// TIA Portal V15.1 export
// export: Created 2024-06-21T08:41:21.5469996Z, ExportSetting WithDefaults, DisplayName Totally Integrated Automation Portal, DisplayVersion V15.1 Update 5, DisplayName TIA Portal Openness, DisplayVersion V15.1 Update 5, DisplayName SINAMICS Startdrive Advanced, DisplayVersion V15.1, DisplayName G130, G150, S120, S150, SINAMICS MV, S210, DisplayVersion V15.1, DisplayName G110M, G120, G120C, G120D, G120P, DisplayVersion V15.1, DisplayName STEP 7 Professional, DisplayVersion V15.1 Update 5, DisplayName STEP 7 Safety, DisplayVersion V15.1, DisplayName WinCC Professional, DisplayVersion V15.1 Update 5, DisplayName SIMATIC Visualization Architect, DisplayVersion V15.1
FUNCTION "209220ZS01AEAK" : Void   // FC371, FBD
TITLE = 209220ZS01AEAK
{ S7_Optimized_Access := 'TRUE' }
AUTHOR : VCC
VERSION : 0.1
// stored: AutoNumber false, IsIECCheckEnabled false, SetENOAutomatically False, UDAEnableTagReadback false
   VAR_OUTPUT
      O_AlarmA : Bool;   // Alarm A
      O_AlarmB : Bool;   // Alarm B
      O_AlarmC : Bool;   // Alarm C
      O_AlarmD : Bool;   // Alarm D
      O_AlarmABCondition : Bool;   // Alarm AB condition
      H_IAnim : Word;   // For animation of icon
   END_VAR
BEGIN

REGION Network 1: **** --------------------- AE01 --------------------- ****
END_REGION

REGION Network 2: **** 2.2 Alarms - Alarm generation **** AE01E3FS10 // CH1 - 24VDC Fuse - ModeZone220 - Switch / Busnode 220AX01 & 220AS10
   // 24VDC Fuse - ModeZone220 - Switch / Busnode 220AX01 & 220AS10
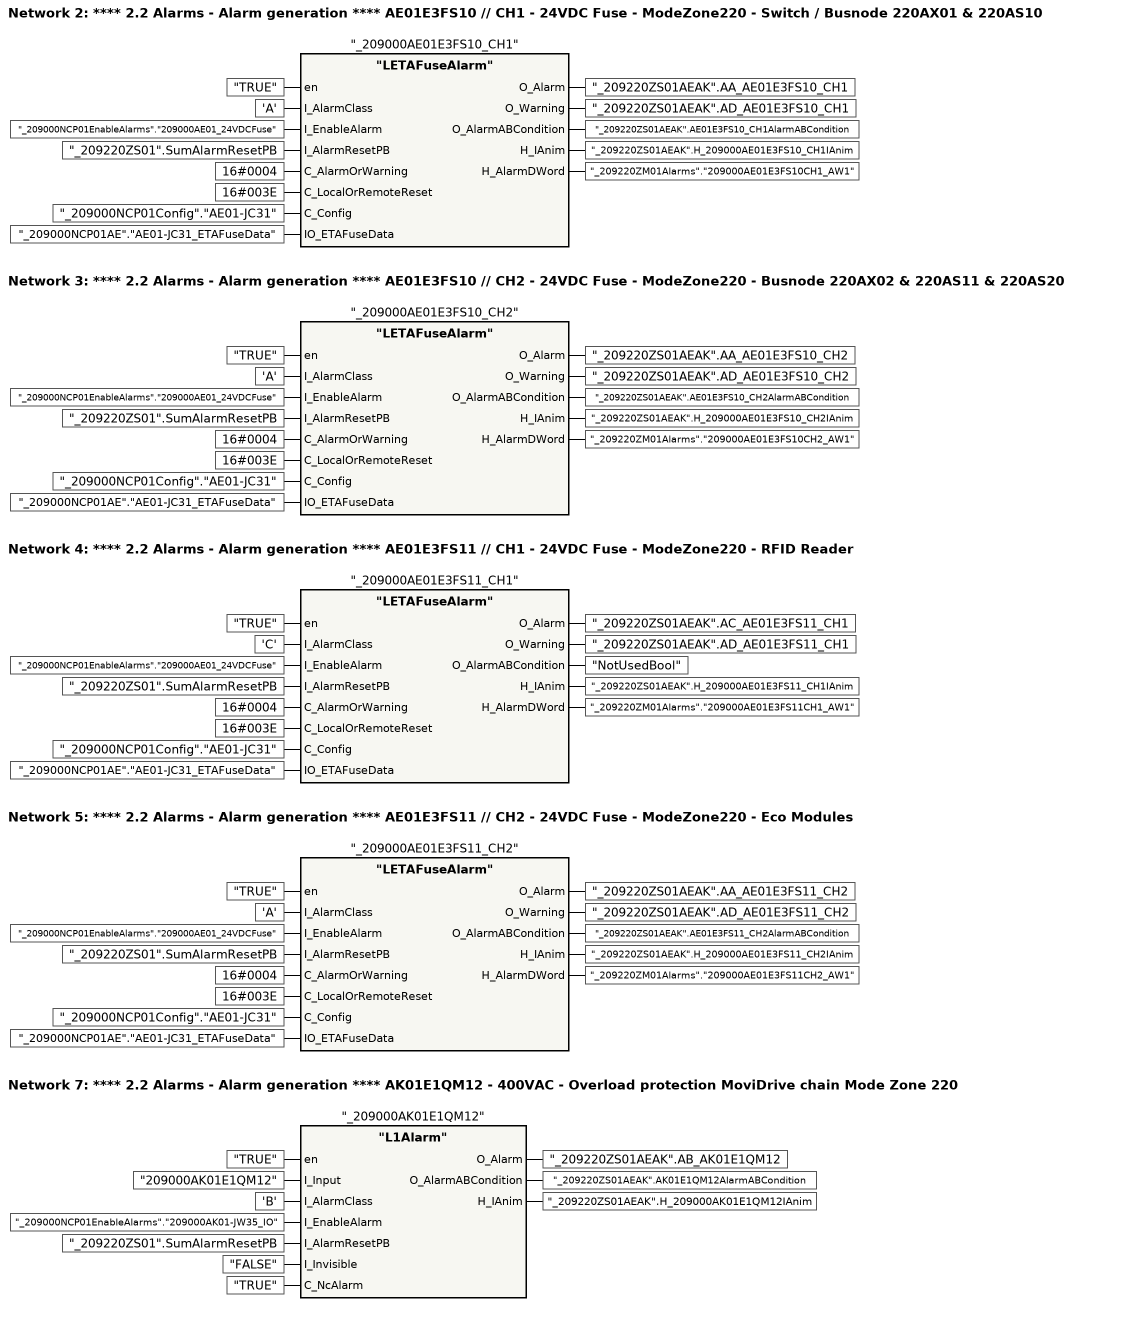
   IF "TRUE" THEN
       "_209000AE01E3FS10_CH1"(I_AlarmClass := 'A',   // "LETAFuseAlarm"
                               I_EnableAlarm := "_209000NCP01EnableAlarms"."209000AE01_24VDCFuse",
                               I_AlarmResetPB := "_209220ZS01".SumAlarmResetPB,
                               C_AlarmOrWarning := 16#0004,
                               C_LocalOrRemoteReset := 16#003E,
                               C_Config := "_209000NCP01Config"."AE01-JC31",
                               IO_ETAFuseData := "_209000NCP01AE"."AE01-JC31_ETAFuseData",
                               O_Alarm => "_209220ZS01AEAK".AA_AE01E3FS10_CH1,
                               O_Warning => "_209220ZS01AEAK".AD_AE01E3FS10_CH1,
                               O_AlarmABCondition => "_209220ZS01AEAK".AE01E3FS10_CH1AlarmABCondition,
                               H_IAnim => "_209220ZS01AEAK".H_209000AE01E3FS10_CH1IAnim,
                               H_AlarmDWord => "_209220ZM01Alarms"."209000AE01E3FS10CH1_AW1");
   END_IF;
END_REGION

REGION Network 3: **** 2.2 Alarms - Alarm generation **** AE01E3FS10 // CH2 - 24VDC Fuse - ModeZone220 - Busnode 220AX02 & 220AS11 & 220AS20
   // 24VDC Fuse - ModeZone220 - Busnode 220AX02 & 220AS11 & 220AS20
   IF "TRUE" THEN
       "_209000AE01E3FS10_CH2"(I_AlarmClass := 'A',   // "LETAFuseAlarm"
                               I_EnableAlarm := "_209000NCP01EnableAlarms"."209000AE01_24VDCFuse",
                               I_AlarmResetPB := "_209220ZS01".SumAlarmResetPB,
                               C_AlarmOrWarning := 16#0004,
                               C_LocalOrRemoteReset := 16#003E,
                               C_Config := "_209000NCP01Config"."AE01-JC31",
                               IO_ETAFuseData := "_209000NCP01AE"."AE01-JC31_ETAFuseData",
                               O_Alarm => "_209220ZS01AEAK".AA_AE01E3FS10_CH2,
                               O_Warning => "_209220ZS01AEAK".AD_AE01E3FS10_CH2,
                               O_AlarmABCondition => "_209220ZS01AEAK".AE01E3FS10_CH2AlarmABCondition,
                               H_IAnim => "_209220ZS01AEAK".H_209000AE01E3FS10_CH2IAnim,
                               H_AlarmDWord => "_209220ZM01Alarms"."209000AE01E3FS10CH2_AW1");
   END_IF;
END_REGION

REGION Network 4: **** 2.2 Alarms - Alarm generation **** AE01E3FS11 // CH1 - 24VDC Fuse - ModeZone220 - RFID Reader
   // 24VDC Fuse - ModeZone220 - RFID Reader
   IF "TRUE" THEN
       "_209000AE01E3FS11_CH1"(I_AlarmClass := 'C',   // "LETAFuseAlarm"
                               I_EnableAlarm := "_209000NCP01EnableAlarms"."209000AE01_24VDCFuse",
                               I_AlarmResetPB := "_209220ZS01".SumAlarmResetPB,
                               C_AlarmOrWarning := 16#0004,
                               C_LocalOrRemoteReset := 16#003E,
                               C_Config := "_209000NCP01Config"."AE01-JC31",
                               IO_ETAFuseData := "_209000NCP01AE"."AE01-JC31_ETAFuseData",
                               O_Alarm => "_209220ZS01AEAK".AC_AE01E3FS11_CH1,
                               O_Warning => "_209220ZS01AEAK".AD_AE01E3FS11_CH1,
                               O_AlarmABCondition => "NotUsedBool",
                               H_IAnim => "_209220ZS01AEAK".H_209000AE01E3FS11_CH1IAnim,
                               H_AlarmDWord => "_209220ZM01Alarms"."209000AE01E3FS11CH1_AW1");
   END_IF;
END_REGION

REGION Network 5: **** 2.2 Alarms - Alarm generation **** AE01E3FS11 // CH2 - 24VDC Fuse - ModeZone220 - Eco Modules
   // 24VDC Fuse - ModeZone220 - Eco Modules
   IF "TRUE" THEN
       "_209000AE01E3FS11_CH2"(I_AlarmClass := 'A',   // "LETAFuseAlarm"
                               I_EnableAlarm := "_209000NCP01EnableAlarms"."209000AE01_24VDCFuse",
                               I_AlarmResetPB := "_209220ZS01".SumAlarmResetPB,
                               C_AlarmOrWarning := 16#0004,
                               C_LocalOrRemoteReset := 16#003E,
                               C_Config := "_209000NCP01Config"."AE01-JC31",
                               IO_ETAFuseData := "_209000NCP01AE"."AE01-JC31_ETAFuseData",
                               O_Alarm => "_209220ZS01AEAK".AA_AE01E3FS11_CH2,
                               O_Warning => "_209220ZS01AEAK".AD_AE01E3FS11_CH2,
                               O_AlarmABCondition => "_209220ZS01AEAK".AE01E3FS11_CH2AlarmABCondition,
                               H_IAnim => "_209220ZS01AEAK".H_209000AE01E3FS11_CH2IAnim,
                               H_AlarmDWord => "_209220ZM01Alarms"."209000AE01E3FS11CH2_AW1");
   END_IF;
END_REGION

REGION Network 6: **** --------------------- AK01 --------------------- ****
END_REGION

REGION Network 7: **** 2.2 Alarms - Alarm generation **** AK01E1QM12 - 400VAC - Overload protection MoviDrive chain Mode Zone 220
   // 400VAC - Overload protection MoviDrive chain Mode Zone 220
   IF "TRUE" THEN
       "_209000AK01E1QM12"(I_Input := "209000AK01E1QM12",   // "L1Alarm"
                           I_AlarmClass := 'B',
                           I_EnableAlarm := "_209000NCP01EnableAlarms"."209000AK01-JW35_IO",
                           I_AlarmResetPB := "_209220ZS01".SumAlarmResetPB,
                           I_Invisible := "FALSE",
                           C_NcAlarm := "TRUE",
                           O_Alarm => "_209220ZS01AEAK".AB_AK01E1QM12,
                           O_AlarmABCondition => "_209220ZS01AEAK".AK01E1QM12AlarmABCondition,
                           H_IAnim => "_209220ZS01AEAK".H_209000AK01E1QM12IAnim);
   END_IF;
END_REGION

REGION Network 8: **** 2.2 Alarms - Alarm generation **** AK01E1QM13 - 400VAC - Overload protection MoviFit chain Mode Zone 220
   // 400VAC - Overload protection MoviFit chain Mode Zone 220
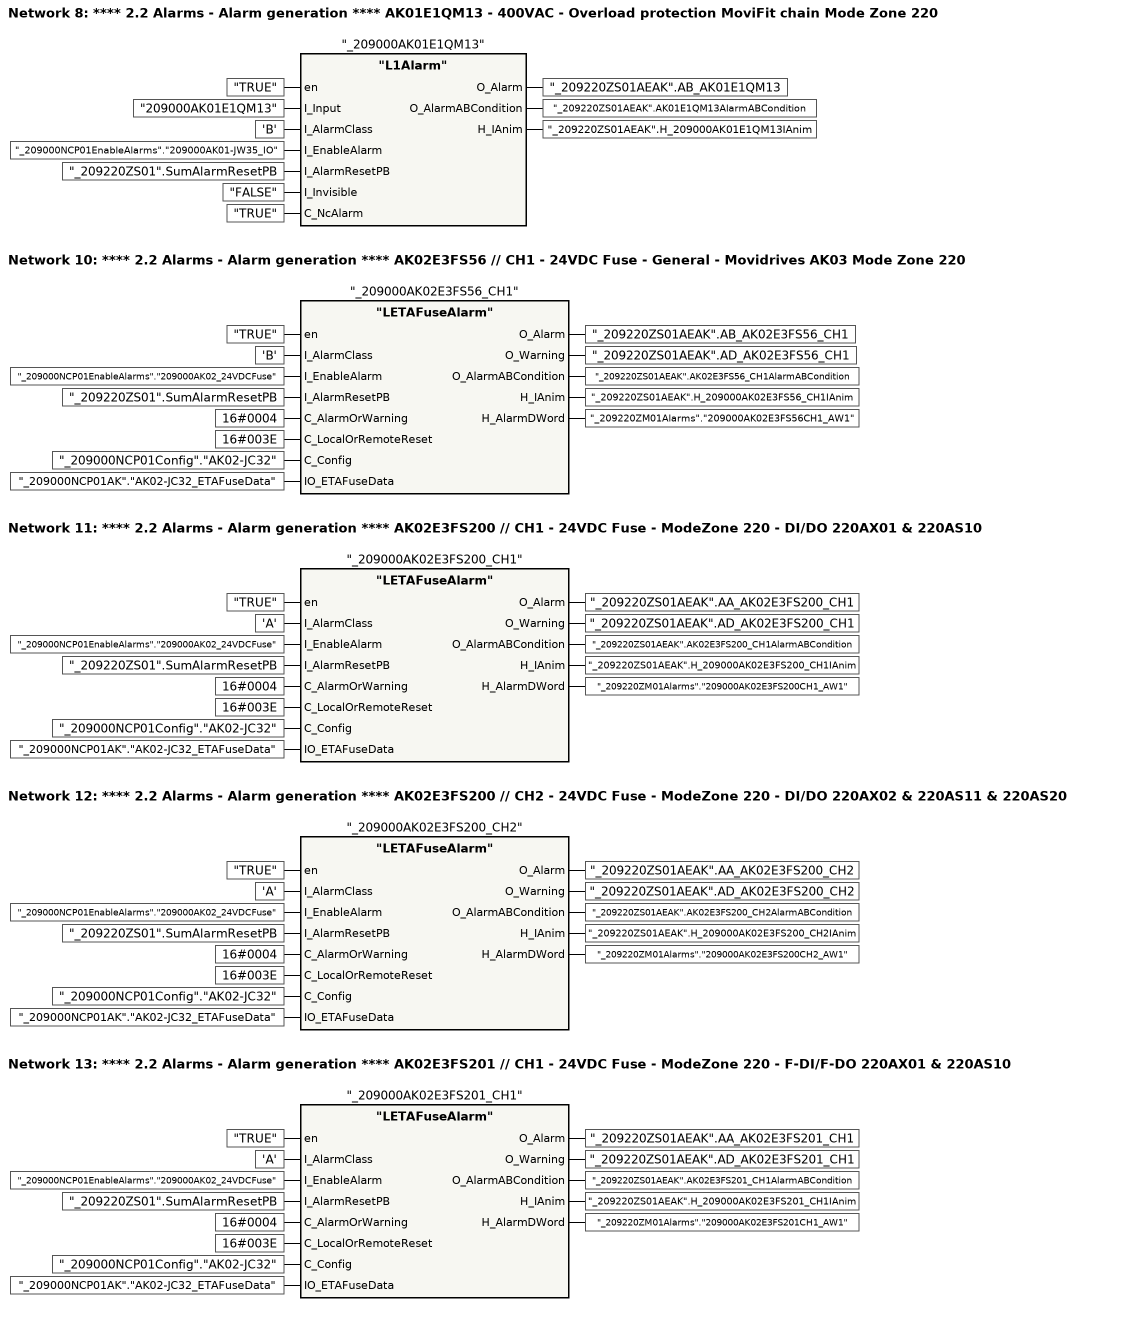
   IF "TRUE" THEN
       "_209000AK01E1QM13"(I_Input := "209000AK01E1QM13",   // "L1Alarm"
                           I_AlarmClass := 'B',
                           I_EnableAlarm := "_209000NCP01EnableAlarms"."209000AK01-JW35_IO",
                           I_AlarmResetPB := "_209220ZS01".SumAlarmResetPB,
                           I_Invisible := "FALSE",
                           C_NcAlarm := "TRUE",
                           O_Alarm => "_209220ZS01AEAK".AB_AK01E1QM13,
                           O_AlarmABCondition => "_209220ZS01AEAK".AK01E1QM13AlarmABCondition,
                           H_IAnim => "_209220ZS01AEAK".H_209000AK01E1QM13IAnim);
   END_IF;
END_REGION

REGION Network 9: **** --------------------- AK02 --------------------- ****
END_REGION

REGION Network 10: **** 2.2 Alarms - Alarm generation **** AK02E3FS56 // CH1 - 24VDC Fuse - General - Movidrives AK03 Mode Zone 220
   // 24VDC Fuse - General - Movidrives AK03 Mode Zone 220
   IF "TRUE" THEN
       "_209000AK02E3FS56_CH1"(I_AlarmClass := 'B',   // "LETAFuseAlarm"
                               I_EnableAlarm := "_209000NCP01EnableAlarms"."209000AK02_24VDCFuse",
                               I_AlarmResetPB := "_209220ZS01".SumAlarmResetPB,
                               C_AlarmOrWarning := 16#0004,
                               C_LocalOrRemoteReset := 16#003E,
                               C_Config := "_209000NCP01Config"."AK02-JC32",
                               IO_ETAFuseData := "_209000NCP01AK"."AK02-JC32_ETAFuseData",
                               O_Alarm => "_209220ZS01AEAK".AB_AK02E3FS56_CH1,
                               O_Warning => "_209220ZS01AEAK".AD_AK02E3FS56_CH1,
                               O_AlarmABCondition => "_209220ZS01AEAK".AK02E3FS56_CH1AlarmABCondition,
                               H_IAnim => "_209220ZS01AEAK".H_209000AK02E3FS56_CH1IAnim,
                               H_AlarmDWord => "_209220ZM01Alarms"."209000AK02E3FS56CH1_AW1");
   END_IF;
END_REGION

REGION Network 11: **** 2.2 Alarms - Alarm generation **** AK02E3FS200 // CH1 - 24VDC Fuse - ModeZone 220 - DI/DO 220AX01 & 220AS10
   // 24VDC Fuse - ModeZone 220 - DI/DO 220AX01 & 220AS10
   IF "TRUE" THEN
       "_209000AK02E3FS200_CH1"(I_AlarmClass := 'A',   // "LETAFuseAlarm"
                               I_EnableAlarm := "_209000NCP01EnableAlarms"."209000AK02_24VDCFuse",
                               I_AlarmResetPB := "_209220ZS01".SumAlarmResetPB,
                               C_AlarmOrWarning := 16#0004,
                               C_LocalOrRemoteReset := 16#003E,
                               C_Config := "_209000NCP01Config"."AK02-JC32",
                               IO_ETAFuseData := "_209000NCP01AK"."AK02-JC32_ETAFuseData",
                               O_Alarm => "_209220ZS01AEAK".AA_AK02E3FS200_CH1,
                               O_Warning => "_209220ZS01AEAK".AD_AK02E3FS200_CH1,
                               O_AlarmABCondition => "_209220ZS01AEAK".AK02E3FS200_CH1AlarmABCondition,
                               H_IAnim => "_209220ZS01AEAK".H_209000AK02E3FS200_CH1IAnim,
                               H_AlarmDWord => "_209220ZM01Alarms"."209000AK02E3FS200CH1_AW1");
   END_IF;
END_REGION

REGION Network 12: **** 2.2 Alarms - Alarm generation **** AK02E3FS200 // CH2 - 24VDC Fuse - ModeZone 220 - DI/DO 220AX02 & 220AS11 & 220AS20
   // 24VDC Fuse - ModeZone 220 - DI/DO 220AX02 & 220AS11 & 220AS20
   IF "TRUE" THEN
       "_209000AK02E3FS200_CH2"(I_AlarmClass := 'A',   // "LETAFuseAlarm"
                               I_EnableAlarm := "_209000NCP01EnableAlarms"."209000AK02_24VDCFuse",
                               I_AlarmResetPB := "_209220ZS01".SumAlarmResetPB,
                               C_AlarmOrWarning := 16#0004,
                               C_LocalOrRemoteReset := 16#003E,
                               C_Config := "_209000NCP01Config"."AK02-JC32",
                               IO_ETAFuseData := "_209000NCP01AK"."AK02-JC32_ETAFuseData",
                               O_Alarm => "_209220ZS01AEAK".AA_AK02E3FS200_CH2,
                               O_Warning => "_209220ZS01AEAK".AD_AK02E3FS200_CH2,
                               O_AlarmABCondition => "_209220ZS01AEAK".AK02E3FS200_CH2AlarmABCondition,
                               H_IAnim => "_209220ZS01AEAK".H_209000AK02E3FS200_CH2IAnim,
                               H_AlarmDWord => "_209220ZM01Alarms"."209000AK02E3FS200CH2_AW1");
   END_IF;
END_REGION

REGION Network 13: **** 2.2 Alarms - Alarm generation **** AK02E3FS201 // CH1 - 24VDC Fuse - ModeZone 220 - F-DI/F-DO 220AX01 & 220AS10
   // 24VDC Fuse - ModeZone 220 - F-DI/F-DO 220AX01 & 220AS10
   IF "TRUE" THEN
       "_209000AK02E3FS201_CH1"(I_AlarmClass := 'A',   // "LETAFuseAlarm"
                               I_EnableAlarm := "_209000NCP01EnableAlarms"."209000AK02_24VDCFuse",
                               I_AlarmResetPB := "_209220ZS01".SumAlarmResetPB,
                               C_AlarmOrWarning := 16#0004,
                               C_LocalOrRemoteReset := 16#003E,
                               C_Config := "_209000NCP01Config"."AK02-JC32",
                               IO_ETAFuseData := "_209000NCP01AK"."AK02-JC32_ETAFuseData",
                               O_Alarm => "_209220ZS01AEAK".AA_AK02E3FS201_CH1,
                               O_Warning => "_209220ZS01AEAK".AD_AK02E3FS201_CH1,
                               O_AlarmABCondition => "_209220ZS01AEAK".AK02E3FS201_CH1AlarmABCondition,
                               H_IAnim => "_209220ZS01AEAK".H_209000AK02E3FS201_CH1IAnim,
                               H_AlarmDWord => "_209220ZM01Alarms"."209000AK02E3FS201CH1_AW1");
   END_IF;
END_REGION

REGION Network 14: **** 2.2 Alarms - Alarm generation **** AK02E3FS201 // CH2 - 24VDC Fuse - ModeZone 220 - F-DI/F-DO 220AX02 & 220AS11 & 220AS20
   // 24VDC Fuse - ModeZone 220 - F-DI/F-DO 220AX02 & 220AS11 & 220AS20
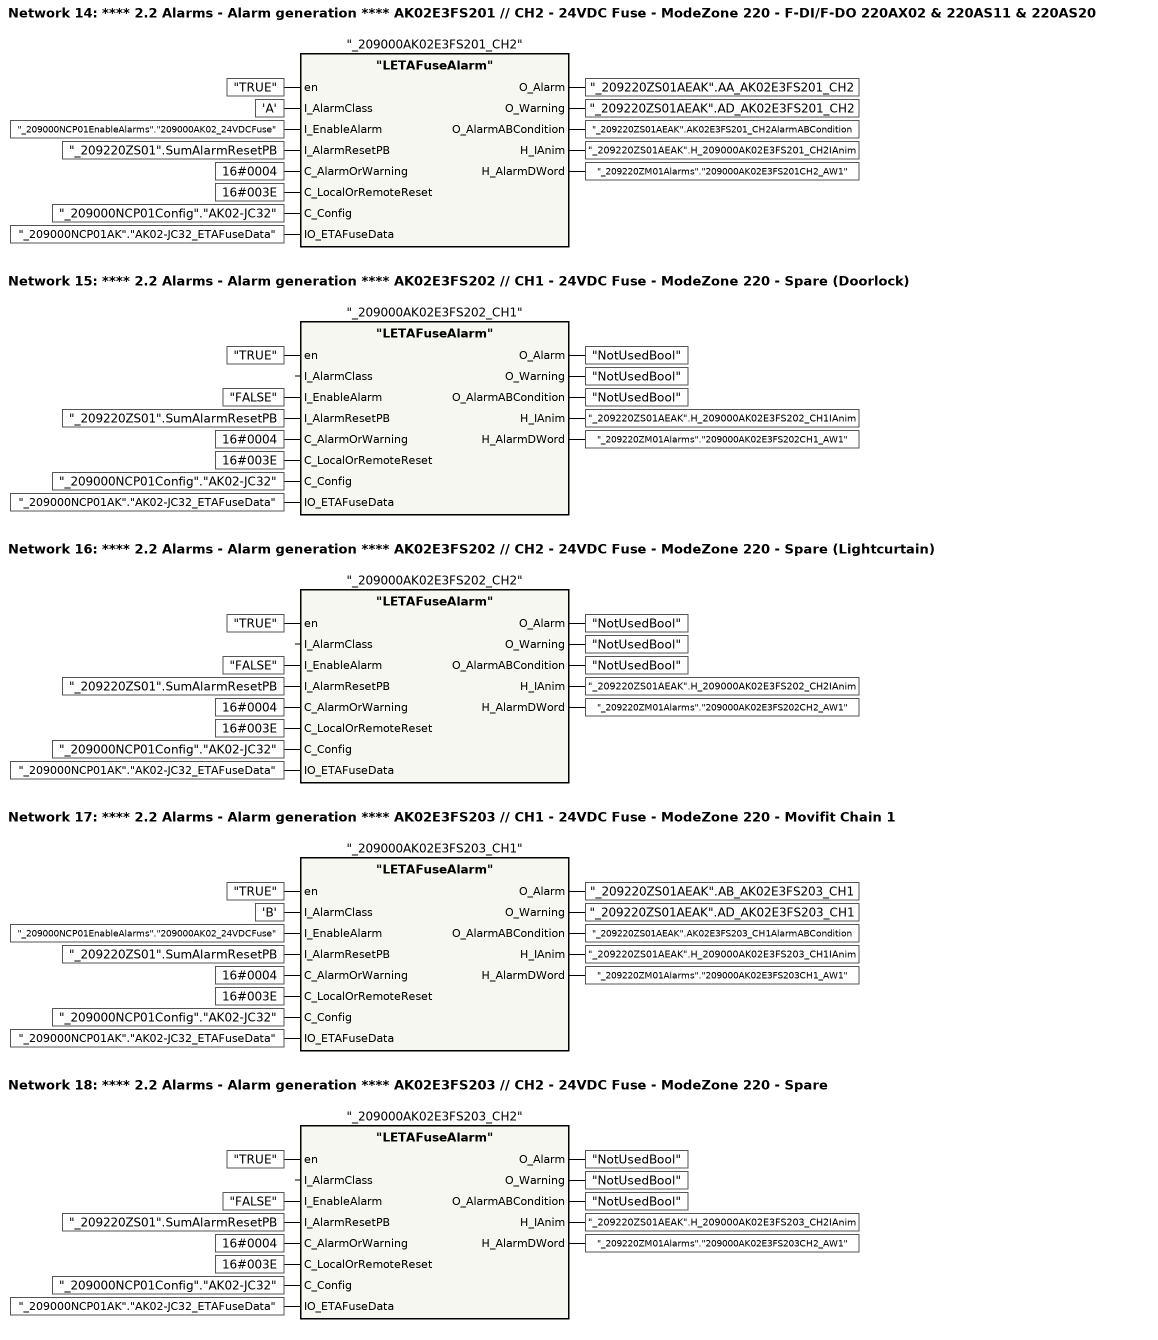
   IF "TRUE" THEN
       "_209000AK02E3FS201_CH2"(I_AlarmClass := 'A',   // "LETAFuseAlarm"
                               I_EnableAlarm := "_209000NCP01EnableAlarms"."209000AK02_24VDCFuse",
                               I_AlarmResetPB := "_209220ZS01".SumAlarmResetPB,
                               C_AlarmOrWarning := 16#0004,
                               C_LocalOrRemoteReset := 16#003E,
                               C_Config := "_209000NCP01Config"."AK02-JC32",
                               IO_ETAFuseData := "_209000NCP01AK"."AK02-JC32_ETAFuseData",
                               O_Alarm => "_209220ZS01AEAK".AA_AK02E3FS201_CH2,
                               O_Warning => "_209220ZS01AEAK".AD_AK02E3FS201_CH2,
                               O_AlarmABCondition => "_209220ZS01AEAK".AK02E3FS201_CH2AlarmABCondition,
                               H_IAnim => "_209220ZS01AEAK".H_209000AK02E3FS201_CH2IAnim,
                               H_AlarmDWord => "_209220ZM01Alarms"."209000AK02E3FS201CH2_AW1");
   END_IF;
END_REGION

REGION Network 15: **** 2.2 Alarms - Alarm generation **** AK02E3FS202 // CH1 - 24VDC Fuse - ModeZone 220 - Spare (Doorlock)
   // 24VDC Fuse - ModeZone 220 - Spare (Doorlock)
   IF "TRUE" THEN
       "_209000AK02E3FS202_CH1"(I_EnableAlarm := "FALSE",   // "LETAFuseAlarm"
                               I_AlarmResetPB := "_209220ZS01".SumAlarmResetPB,
                               C_AlarmOrWarning := 16#0004,
                               C_LocalOrRemoteReset := 16#003E,
                               C_Config := "_209000NCP01Config"."AK02-JC32",
                               IO_ETAFuseData := "_209000NCP01AK"."AK02-JC32_ETAFuseData",
                               O_Alarm => "NotUsedBool",
                               O_Warning => "NotUsedBool",
                               O_AlarmABCondition => "NotUsedBool",
                               H_IAnim => "_209220ZS01AEAK".H_209000AK02E3FS202_CH1IAnim,
                               H_AlarmDWord => "_209220ZM01Alarms"."209000AK02E3FS202CH1_AW1");
   END_IF;
END_REGION

REGION Network 16: **** 2.2 Alarms - Alarm generation **** AK02E3FS202 // CH2 - 24VDC Fuse - ModeZone 220 - Spare (Lightcurtain)
   // 24VDC Fuse - ModeZone 220 - Spare (Lightcurtain)
   IF "TRUE" THEN
       "_209000AK02E3FS202_CH2"(I_EnableAlarm := "FALSE",   // "LETAFuseAlarm"
                               I_AlarmResetPB := "_209220ZS01".SumAlarmResetPB,
                               C_AlarmOrWarning := 16#0004,
                               C_LocalOrRemoteReset := 16#003E,
                               C_Config := "_209000NCP01Config"."AK02-JC32",
                               IO_ETAFuseData := "_209000NCP01AK"."AK02-JC32_ETAFuseData",
                               O_Alarm => "NotUsedBool",
                               O_Warning => "NotUsedBool",
                               O_AlarmABCondition => "NotUsedBool",
                               H_IAnim => "_209220ZS01AEAK".H_209000AK02E3FS202_CH2IAnim,
                               H_AlarmDWord => "_209220ZM01Alarms"."209000AK02E3FS202CH2_AW1");
   END_IF;
END_REGION

REGION Network 17: **** 2.2 Alarms - Alarm generation **** AK02E3FS203 // CH1 - 24VDC Fuse - ModeZone 220 - Movifit Chain 1
   // 24VDC Fuse - ModeZone 220 - Movifit Chain 1
   IF "TRUE" THEN
       "_209000AK02E3FS203_CH1"(I_AlarmClass := 'B',   // "LETAFuseAlarm"
                               I_EnableAlarm := "_209000NCP01EnableAlarms"."209000AK02_24VDCFuse",
                               I_AlarmResetPB := "_209220ZS01".SumAlarmResetPB,
                               C_AlarmOrWarning := 16#0004,
                               C_LocalOrRemoteReset := 16#003E,
                               C_Config := "_209000NCP01Config"."AK02-JC32",
                               IO_ETAFuseData := "_209000NCP01AK"."AK02-JC32_ETAFuseData",
                               O_Alarm => "_209220ZS01AEAK".AB_AK02E3FS203_CH1,
                               O_Warning => "_209220ZS01AEAK".AD_AK02E3FS203_CH1,
                               O_AlarmABCondition => "_209220ZS01AEAK".AK02E3FS203_CH1AlarmABCondition,
                               H_IAnim => "_209220ZS01AEAK".H_209000AK02E3FS203_CH1IAnim,
                               H_AlarmDWord => "_209220ZM01Alarms"."209000AK02E3FS203CH1_AW1");
   END_IF;
END_REGION

REGION Network 18: **** 2.2 Alarms - Alarm generation **** AK02E3FS203 // CH2 - 24VDC Fuse - ModeZone 220 - Spare
   // 24VDC Fuse - ModeZone 220 - Spare
   IF "TRUE" THEN
       "_209000AK02E3FS203_CH2"(I_EnableAlarm := "FALSE",   // "LETAFuseAlarm"
                               I_AlarmResetPB := "_209220ZS01".SumAlarmResetPB,
                               C_AlarmOrWarning := 16#0004,
                               C_LocalOrRemoteReset := 16#003E,
                               C_Config := "_209000NCP01Config"."AK02-JC32",
                               IO_ETAFuseData := "_209000NCP01AK"."AK02-JC32_ETAFuseData",
                               O_Alarm => "NotUsedBool",
                               O_Warning => "NotUsedBool",
                               O_AlarmABCondition => "NotUsedBool",
                               H_IAnim => "_209220ZS01AEAK".H_209000AK02E3FS203_CH2IAnim,
                               H_AlarmDWord => "_209220ZM01Alarms"."209000AK02E3FS203CH2_AW1");
   END_IF;
END_REGION

REGION Network 19: **** --------------------- AK04 --------------------- ****
END_REGION

REGION Network 20: **** 2.2 Alarms - Alarm generation **** AK04E1QM140 - 400VAC - Overload protection Brake Resistor 209220CR21
   // 400VAC - Overload protection Brake Resistor 209220CR21
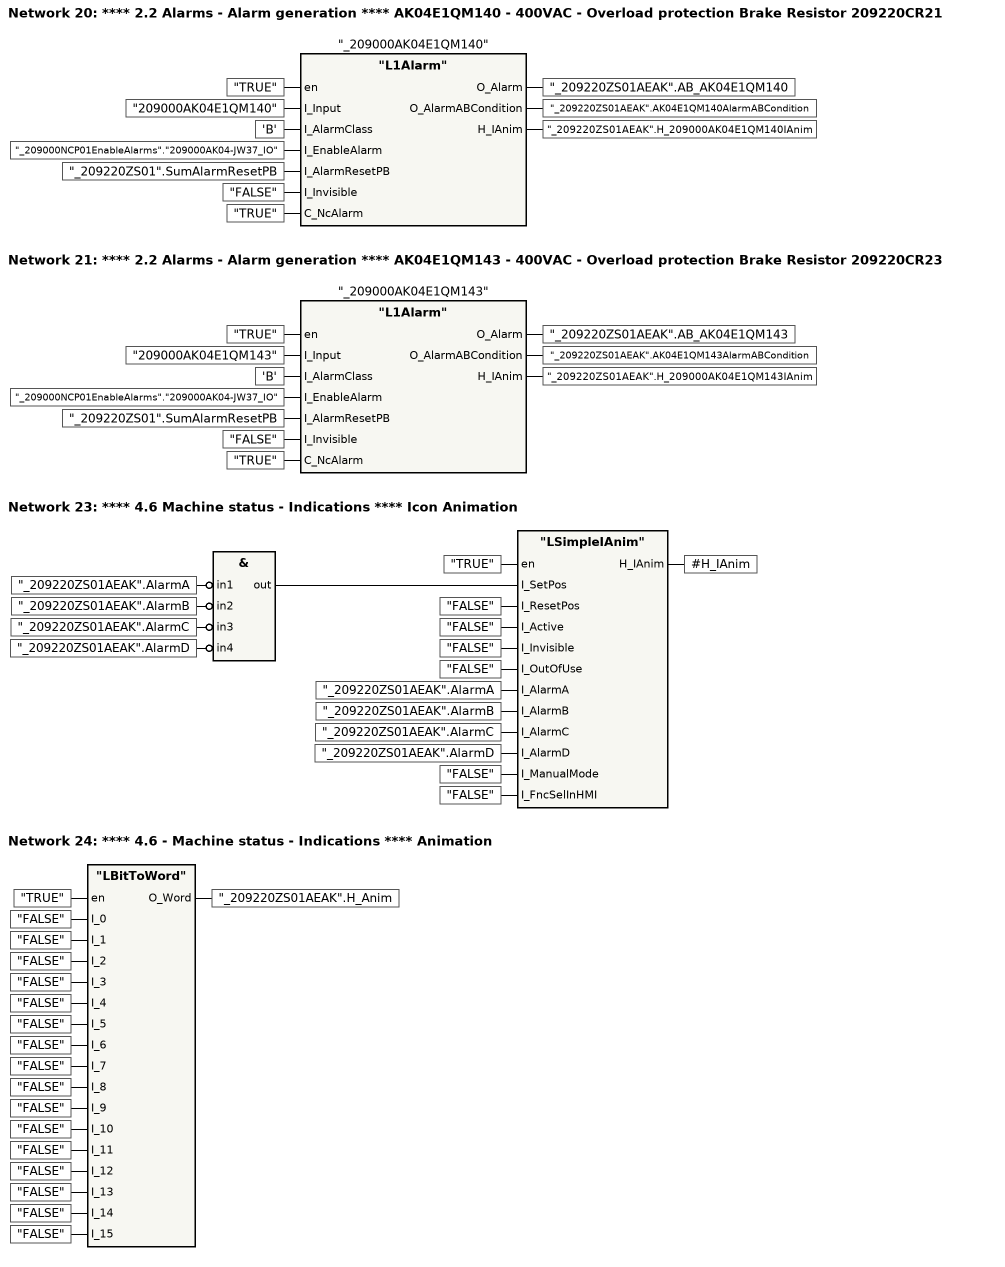
   IF "TRUE" THEN
       "_209000AK04E1QM140"(I_Input := "209000AK04E1QM140",   // "L1Alarm"
                            I_AlarmClass := 'B',
                            I_EnableAlarm := "_209000NCP01EnableAlarms"."209000AK04-JW37_IO",
                            I_AlarmResetPB := "_209220ZS01".SumAlarmResetPB,
                            I_Invisible := "FALSE",
                            C_NcAlarm := "TRUE",
                            O_Alarm => "_209220ZS01AEAK".AB_AK04E1QM140,
                            O_AlarmABCondition => "_209220ZS01AEAK".AK04E1QM140AlarmABCondition,
                            H_IAnim => "_209220ZS01AEAK".H_209000AK04E1QM140IAnim);
   END_IF;
END_REGION

REGION Network 21: **** 2.2 Alarms - Alarm generation **** AK04E1QM143 - 400VAC - Overload protection Brake Resistor 209220CR23
   // 400VAC - Overload protection Brake Resistor 209220CR23
   IF "TRUE" THEN
       "_209000AK04E1QM143"(I_Input := "209000AK04E1QM143",   // "L1Alarm"
                            I_AlarmClass := 'B',
                            I_EnableAlarm := "_209000NCP01EnableAlarms"."209000AK04-JW37_IO",
                            I_AlarmResetPB := "_209220ZS01".SumAlarmResetPB,
                            I_Invisible := "FALSE",
                            C_NcAlarm := "TRUE",
                            O_Alarm => "_209220ZS01AEAK".AB_AK04E1QM143,
                            O_AlarmABCondition => "_209220ZS01AEAK".AK04E1QM143AlarmABCondition,
                            H_IAnim => "_209220ZS01AEAK".H_209000AK04E1QM143IAnim);
   END_IF;
END_REGION

REGION Network 22: **** -------------------------------------------------- ****
END_REGION

REGION Network 23: **** 4.6 Machine status - Indications **** Icon Animation
   // Animation for icon
   IF "TRUE" THEN
       "LSimpleIAnim"(I_SetPos := NOT "_209220ZS01AEAK".AlarmA AND NOT "_209220ZS01AEAK".AlarmB AND NOT "_209220ZS01AEAK".AlarmC AND NOT "_209220ZS01AEAK".AlarmD,
                      I_ResetPos := "FALSE",
                      I_Active := "FALSE",
                      I_Invisible := "FALSE",
                      I_OutOfUse := "FALSE",
                      I_AlarmA := "_209220ZS01AEAK".AlarmA,
                      I_AlarmB := "_209220ZS01AEAK".AlarmB,
                      I_AlarmC := "_209220ZS01AEAK".AlarmC,
                      I_AlarmD := "_209220ZS01AEAK".AlarmD,
                      I_ManualMode := "FALSE",
                      I_FncSelInHMI := "FALSE",
                      H_IAnim => #H_IAnim);
   END_IF;
END_REGION

REGION Network 24: **** 4.6 - Machine status - Indications **** Animation
   // Animation
   IF "TRUE" THEN
       "LBitToWord"(I_0 := "FALSE",
                    I_1 := "FALSE",
                    I_2 := "FALSE",
                    I_3 := "FALSE",
                    I_4 := "FALSE",
                    I_5 := "FALSE",
                    I_6 := "FALSE",
                    I_7 := "FALSE",
                    I_8 := "FALSE",
                    I_9 := "FALSE",
                    I_10 := "FALSE",
                    I_11 := "FALSE",
                    I_12 := "FALSE",
                    I_13 := "FALSE",
                    I_14 := "FALSE",
                    I_15 := "FALSE",
                    O_Word => "_209220ZS01AEAK".H_Anim);
   END_IF;
END_REGION

NETWORK
TITLE = **** 4.6 - Machine Status - Indications **** Animation DB number
// DB number
      OPN   "_209220ZS01AEAK";
      L     DBNO;
      T     "_209220ZS01AEAK".H_DBnr;

REGION Network 26: **** 9 - Alarm Summary **** Alarm AB condition
   // Alarm AB condition
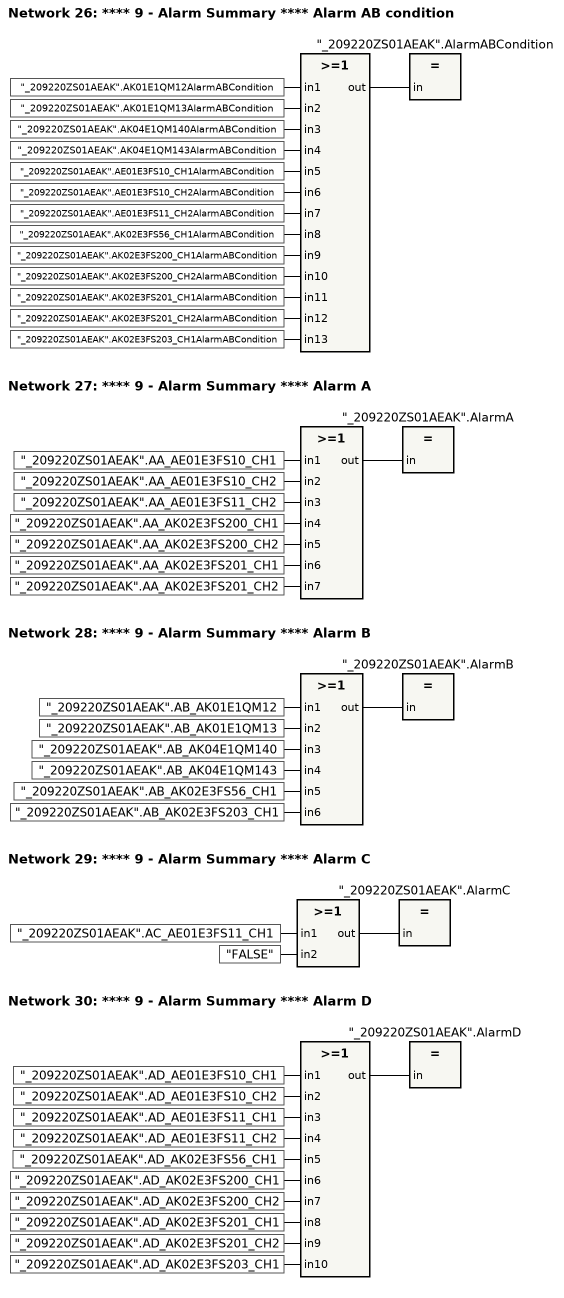
   "_209220ZS01AEAK".AlarmABCondition := "_209220ZS01AEAK".AK01E1QM12AlarmABCondition OR "_209220ZS01AEAK".AK01E1QM13AlarmABCondition OR "_209220ZS01AEAK".AK04E1QM140AlarmABCondition OR "_209220ZS01AEAK".AK04E1QM143AlarmABCondition OR "_209220ZS01AEAK".AE01E3FS10_CH1AlarmABCondition OR "_209220ZS01AEAK".AE01E3FS10_CH2AlarmABCondition OR "_209220ZS01AEAK".AE01E3FS11_CH2AlarmABCondition OR "_209220ZS01AEAK".AK02E3FS56_CH1AlarmABCondition OR "_209220ZS01AEAK".AK02E3FS200_CH1AlarmABCondition OR "_209220ZS01AEAK".AK02E3FS200_CH2AlarmABCondition OR "_209220ZS01AEAK".AK02E3FS201_CH1AlarmABCondition OR "_209220ZS01AEAK".AK02E3FS201_CH2AlarmABCondition OR "_209220ZS01AEAK".AK02E3FS203_CH1AlarmABCondition;
END_REGION

REGION Network 27: **** 9 - Alarm Summary **** Alarm A
   // Summary of alarms A
   "_209220ZS01AEAK".AlarmA := "_209220ZS01AEAK".AA_AE01E3FS10_CH1 OR "_209220ZS01AEAK".AA_AE01E3FS10_CH2 OR "_209220ZS01AEAK".AA_AE01E3FS11_CH2 OR "_209220ZS01AEAK".AA_AK02E3FS200_CH1 OR "_209220ZS01AEAK".AA_AK02E3FS200_CH2 OR "_209220ZS01AEAK".AA_AK02E3FS201_CH1 OR "_209220ZS01AEAK".AA_AK02E3FS201_CH2;
END_REGION

REGION Network 28: **** 9 - Alarm Summary **** Alarm B
   // Summary of alarms B
   "_209220ZS01AEAK".AlarmB := "_209220ZS01AEAK".AB_AK01E1QM12 OR "_209220ZS01AEAK".AB_AK01E1QM13 OR "_209220ZS01AEAK".AB_AK04E1QM140 OR "_209220ZS01AEAK".AB_AK04E1QM143 OR "_209220ZS01AEAK".AB_AK02E3FS56_CH1 OR "_209220ZS01AEAK".AB_AK02E3FS203_CH1;
END_REGION

REGION Network 29: **** 9 - Alarm Summary **** Alarm C
   // Summary of alarms C
   "_209220ZS01AEAK".AlarmC := "_209220ZS01AEAK".AC_AE01E3FS11_CH1 OR "FALSE";
END_REGION

REGION Network 30: **** 9 - Alarm Summary **** Alarm D
   // Summary of alarms D
   "_209220ZS01AEAK".AlarmD := "_209220ZS01AEAK".AD_AE01E3FS10_CH1 OR "_209220ZS01AEAK".AD_AE01E3FS10_CH2 OR "_209220ZS01AEAK".AD_AE01E3FS11_CH1 OR "_209220ZS01AEAK".AD_AE01E3FS11_CH2 OR "_209220ZS01AEAK".AD_AK02E3FS56_CH1 OR "_209220ZS01AEAK".AD_AK02E3FS200_CH1 OR "_209220ZS01AEAK".AD_AK02E3FS200_CH2 OR "_209220ZS01AEAK".AD_AK02E3FS201_CH1 OR "_209220ZS01AEAK".AD_AK02E3FS201_CH2 OR "_209220ZS01AEAK".AD_AK02E3FS203_CH1;
END_REGION

REGION Network 31: **** 9.1 - Alarm Output **** Alarm AB condition
   // Alarm AB condition
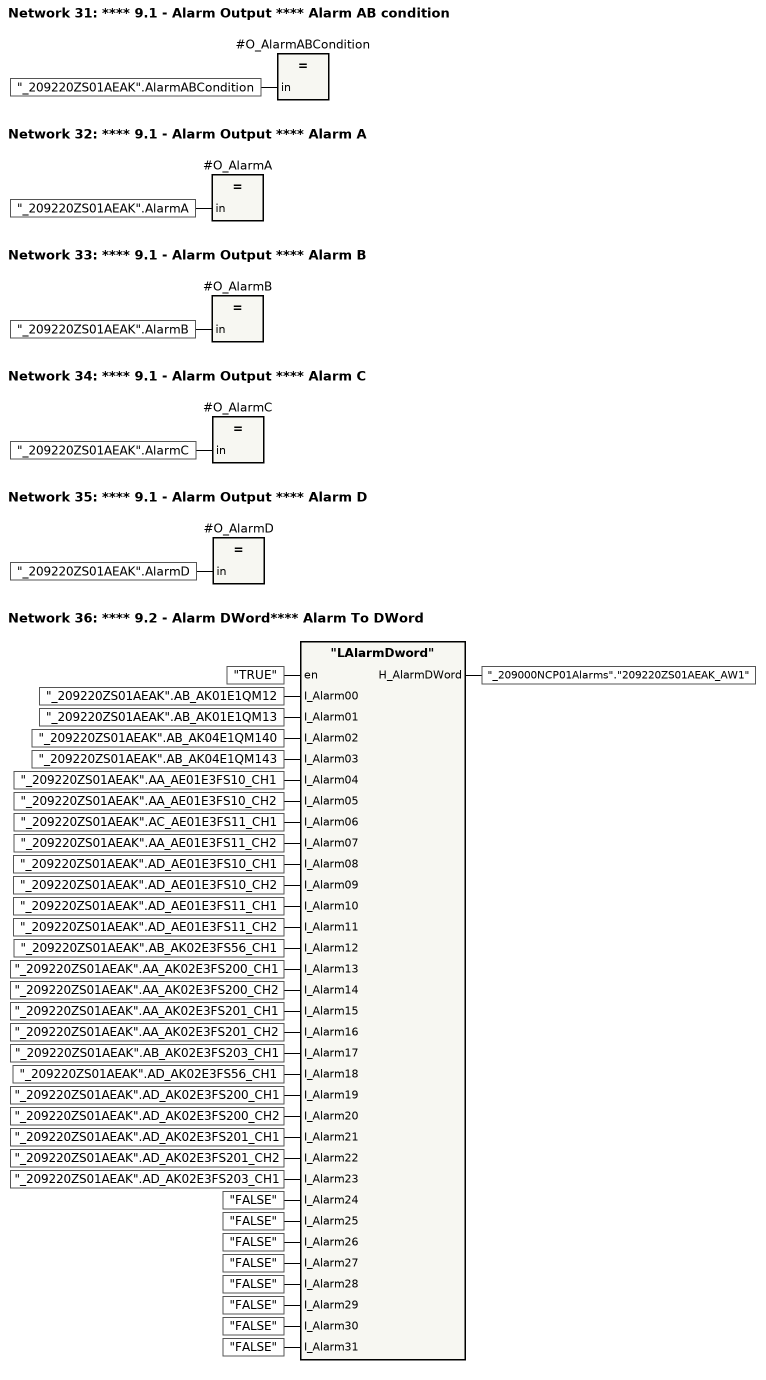
   #O_AlarmABCondition := "_209220ZS01AEAK".AlarmABCondition;
END_REGION

REGION Network 32: **** 9.1 - Alarm Output **** Alarm A
   // Summary of alarms A
   #O_AlarmA := "_209220ZS01AEAK".AlarmA;
END_REGION

REGION Network 33: **** 9.1 - Alarm Output **** Alarm B
   // Summary of alarms B
   #O_AlarmB := "_209220ZS01AEAK".AlarmB;
END_REGION

REGION Network 34: **** 9.1 - Alarm Output **** Alarm C
   // Summary of alarms C
   #O_AlarmC := "_209220ZS01AEAK".AlarmC;
END_REGION

REGION Network 35: **** 9.1 - Alarm Output **** Alarm D
   // Summary of alarms D
   #O_AlarmD := "_209220ZS01AEAK".AlarmD;
END_REGION

REGION Network 36: **** 9.2 - Alarm DWord**** Alarm To DWord
   // Alarm Word
   IF "TRUE" THEN
       "LAlarmDword"(I_Alarm00 := "_209220ZS01AEAK".AB_AK01E1QM12,
                     I_Alarm01 := "_209220ZS01AEAK".AB_AK01E1QM13,
                     I_Alarm02 := "_209220ZS01AEAK".AB_AK04E1QM140,
                     I_Alarm03 := "_209220ZS01AEAK".AB_AK04E1QM143,
                     I_Alarm04 := "_209220ZS01AEAK".AA_AE01E3FS10_CH1,
                     I_Alarm05 := "_209220ZS01AEAK".AA_AE01E3FS10_CH2,
                     I_Alarm06 := "_209220ZS01AEAK".AC_AE01E3FS11_CH1,
                     I_Alarm07 := "_209220ZS01AEAK".AA_AE01E3FS11_CH2,
                     I_Alarm08 := "_209220ZS01AEAK".AD_AE01E3FS10_CH1,
                     I_Alarm09 := "_209220ZS01AEAK".AD_AE01E3FS10_CH2,
                     I_Alarm10 := "_209220ZS01AEAK".AD_AE01E3FS11_CH1,
                     I_Alarm11 := "_209220ZS01AEAK".AD_AE01E3FS11_CH2,
                     I_Alarm12 := "_209220ZS01AEAK".AB_AK02E3FS56_CH1,
                     I_Alarm13 := "_209220ZS01AEAK".AA_AK02E3FS200_CH1,
                     I_Alarm14 := "_209220ZS01AEAK".AA_AK02E3FS200_CH2,
                     I_Alarm15 := "_209220ZS01AEAK".AA_AK02E3FS201_CH1,
                     I_Alarm16 := "_209220ZS01AEAK".AA_AK02E3FS201_CH2,
                     I_Alarm17 := "_209220ZS01AEAK".AB_AK02E3FS203_CH1,
                     I_Alarm18 := "_209220ZS01AEAK".AD_AK02E3FS56_CH1,
                     I_Alarm19 := "_209220ZS01AEAK".AD_AK02E3FS200_CH1,
                     I_Alarm20 := "_209220ZS01AEAK".AD_AK02E3FS200_CH2,
                     I_Alarm21 := "_209220ZS01AEAK".AD_AK02E3FS201_CH1,
                     I_Alarm22 := "_209220ZS01AEAK".AD_AK02E3FS201_CH2,
                     I_Alarm23 := "_209220ZS01AEAK".AD_AK02E3FS203_CH1,
                     I_Alarm24 := "FALSE",
                     I_Alarm25 := "FALSE",
                     I_Alarm26 := "FALSE",
                     I_Alarm27 := "FALSE",
                     I_Alarm28 := "FALSE",
                     I_Alarm29 := "FALSE",
                     I_Alarm30 := "FALSE",
                     I_Alarm31 := "FALSE",
                     H_AlarmDWord => "_209000NCP01Alarms"."209220ZS01AEAK_AW1");
   END_IF;
END_REGION
END_FUNCTION
